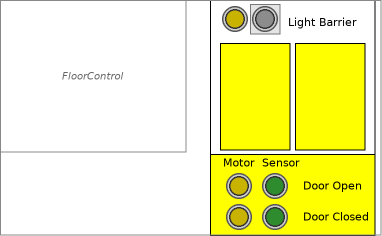
VISUALIZATION Floor  // 382x236
VAR_IN_OUT
	Color 			: DWORD;
	LED_Up	 		: BOOL;
	LED_Down		: BOOL;
	FloorNumber 	: INT;
	BtnLed	 		: ARRAY[1..6] OF BOOL;;
	Btn				: ARRAY[1..6] OF BOOL;
	LB	 			: BOOL;
	LED_DoorOpen 	: BOOL;
	LED_DoorClosed	: BOOL;
	PositionDoor	: REAL;
	M_Open 			: BOOL;
	M_Close			: BOOL;
END_VAR
    Frame (0,0 186x152)
        shows FloorControl(LED_Up := LED_Up, LED_Down := LED_Down, FloorNumber := FloorNumber, BtnLed := BtnLed, Btn := Btn)
    Rectangle (210,0 165x236)
    Rectangle (210,154 165x82), colour variable: Color
    Rectangle (295,43 70x107), colour variable: Color
        p3560616238: (40/100.0*PositionDoor)
    Rectangle (220,43 70x107), colour variable: Color
        p3560616238: -(40/100.0*PositionDoor)
    Lamp1 (260,171 30x30), variable: LED_DoorOpen, style: Lamp-Lamp1-Green
    Lamp1 (260,202 30x30), variable: LED_DoorClosed, style: Lamp-Lamp1-Green
    Label (300,171 82x30), "Door Open"
    Label (300,202 82x30), "Door Closed"
    Label (285,11 82x23), "Light Barrier"
    Lamp1 (220,4 30x30), variable: LB, style: Lamp-Lamp1-Yellow
    PushSwitch (250,4 30x30), variable: LB, behaviour: TAP, style: Switch-PushSwitch-Gray
    Lamp1 (224,202 30x30), variable: M_Close, style: Lamp-Lamp1-Yellow
    Lamp1 (224,171 30x30), variable: M_Open, style: Lamp-Lamp1-Yellow
    Label (220,148 41x30), "Motor"
    Label (259,148 41x30), "Sensor"
END_VISUALIZATION

(* stored: Version 1.1.0.1
   Visu Floor: Id {17733648-0a16-4068-98c8-ac3fb543be38} *)
